{attribute 'linkalways'} 
{attribute 'no_explicit_call' := 'This FB is a CLASS and must be accessed using methods or properties'}
{attribute 'enable_dynamic_creation'}
FUNCTION_BLOCK FINAL LT_WORD EXTENDS Node
VAR
	in1 : _WORD(0);
	in2 : _WORD(0);
	out : _BOOL(FALSE);
END_VAR

METHOD PUBLIC Clone : I_Node
VAR
	pNode : POINTER TO LT_WORD;
END_VAR
pNode := __NEW(LT_WORD);
Clone := pNode^;
END_METHOD

METHOD FB_init : BOOL
VAR_INPUT
	bInitRetains : BOOL; // if TRUE, the retain variables are initialized (warm start / cold start)
	bInCopyCode : BOOL;  // if TRUE, the instance afterwards gets moved into the copy code (online change)
END_VAR
AddInput('in1',THIS^.in1);
AddInput('in2',THIS^.in2);
AddOutput('out', THIS^.out);
END_METHOD

METHOD PROTECTED OnExecute
VAR
END_VAR
out.Value := in1.Value < in2.Value;
END_METHOD

END_FUNCTION_BLOCK

(* stored: Version 1.1.0.1, ProductVersion 3.1.4024.15
   POU LT_WORD: Id {b5493792-b43b-4b31-a6e2-220003e7c8b5}, SpecialFunc None
   Folder Constructor: Id {ca29208d-610c-49e3-b711-0f4a6df3fb3e}
   Method Clone: Id {b90c4666-bfd6-4392-a734-432de9149368}
   Method FB_init: Id {0b1536ca-8f1d-40c7-8805-3ab7b0afc787}
   Method OnExecute: Id {fca72258-70b6-4370-8ee1-d516bb913102} *)
